// TIA Portal V18 export
// export: Created 2026-01-09T11:31:55.5781549Z, ExportSetting WithDefaults, DisplayName Totally Integrated Automation Portal, DisplayVersion V18 Update 5, DisplayName TIA Portal Openness, DisplayVersion V18 Update 5, DisplayName TIA Portal Teamcenter Gateway, DisplayVersion V18, DisplayName TIA Portal Version Control Interface, DisplayVersion V18, DisplayName SINAMICS Startdrive Advanced, DisplayVersion V18 SP2 Update 1, DisplayName SINAMICS Startdrive G110M, G120, G120C, G120D, G120P, G115D, DisplayVersion V18 SP2 Update 1, DisplayName SINAMICS Startdrive G130, G150, S120, S150, SINAMICS MV, S210, G220, S200, DisplayVersion V18 SP2 Update 1, DisplayName STEP 7 Professional, DisplayVersion V18 Update 5, DisplayName STEP 7 Safety, DisplayVersion V18, DisplayName WinCC Professional, DisplayVersion V18 Update 5
TagTable "ST350_Stopper"
  ST350_Stopper_InterfaceDB.aDev[1] : ST_Stopper  (PLC tag ST10_Stopper_InterfaceDB.aDev[1], CPU S71500-2PN_TP700, 100 ms)
    TagStructureMember "ReleasePB"
    TagStructureMember "NoClear"
    TagStructureMember "Sensor"
    TagStructureMember "AutoTrg"
    TagStructureMember "Done"
    TagStructureMember "ReleaseFault"
    TagStructureMember "ReachFault"
  ST350_Stopper_InterfaceDB.aDev[2] : ST_Stopper  (PLC tag ST10_Stopper_InterfaceDB.aDev[2], CPU S71500-2PN_TP700, 100 ms)
    TagStructureMember "ReleasePB"
    TagStructureMember "NoClear"
    TagStructureMember "Sensor"
    TagStructureMember "AutoTrg"
    TagStructureMember "Done"
    TagStructureMember "ReleaseFault"
    TagStructureMember "ReachFault"
  ST350_Stopper_InterfaceDB.aDev[3] : ST_Stopper  (PLC tag ST10_Stopper_InterfaceDB.aDev[3], CPU S71500-2PN_TP700, 100 ms)
    TagStructureMember "ReleasePB"
    TagStructureMember "NoClear"
    TagStructureMember "Sensor"
    TagStructureMember "AutoTrg"
    TagStructureMember "Done"
    TagStructureMember "ReleaseFault"
    TagStructureMember "ReachFault"
  ST350_Stopper_InterfaceDB.aDev[4] : ST_Stopper  (PLC tag ST10_Stopper_InterfaceDB.aDev[4], CPU S71500-2PN_TP700, 100 ms)
    TagStructureMember "ReleasePB"
    TagStructureMember "NoClear"
    TagStructureMember "Sensor"
    TagStructureMember "AutoTrg"
    TagStructureMember "Done"
    TagStructureMember "ReleaseFault"
    TagStructureMember "ReachFault"
  ST350_Stopper_InterfaceDB.aDev[5] : ST_Stopper  (PLC tag ST10_Stopper_InterfaceDB.aDev[5], CPU S71500-2PN_TP700, 100 ms)
    TagStructureMember "ReleasePB"
    TagStructureMember "NoClear"
    TagStructureMember "Sensor"
    TagStructureMember "AutoTrg"
    TagStructureMember "Done"
    TagStructureMember "ReleaseFault"
    TagStructureMember "ReachFault"
